Fanuc KAREL source: VREG_FND_POS.kl

PROGRAM T
%NOLOCKGROUP
VAR
 v0 : INTEGER
 v1 : INTEGER
 v2 : INTEGER
 v3 : INTEGER
BEGIN
 VREG_FND_POS(v0, v1, v2, v3)
END T
